FUNCTION_BLOCK CommonRack EXTENDS RunUnitGeneric
VAR_INPUT
END_VAR
VAR_OUTPUT
END_VAR
VAR
	button : POINTER TO RunSignal ;
	//TODO : define a simple output DO or DO - device?
	
	fixer : POINTER TO RunCylinder;
	approx : POINTER TO RunSignal; // approx then lock
	//---------------------------------
	//	Over Fieldbus linked with SCARA
	//---------------------------------
	rackReady AT%Q*: BOOL;
	rackEngaged AT%I*: BOOL;	

	items : ARRAY[0..3] OF defItem;
	//---------------------------------
	//	Internal
	//---------------------------------
	nCounter : INT;
END_VAR
VAR PERSISTENT
	
END_VAR


//Control the working flow of rack

SUPER^();

CASE outputState OF
	eSpecialStates.SLAVE_ENTER_PROCEDURE:
		//rack is empty
		bSerialTransition := fixer^.Execute(eCylinderCommands.COMMAND_A); //relase
		//TODO , set light flicking
	16#201:
		bSerialTransition := approx^.debouncedOn; //wait until rack closed
	16#202:
		//confirmed by hanshaking
		bSerialTransition := button^.debouncedOn;
		//TODO , set light constant on
	16#203:
		bSerialTransition := fixer^.Execute(eCylinderCommands.COMMAND_B); //lock
		IF bSerialTransition THEN
			rackReady := TRUE;
		END_IF
//		NextState := eSpecialStates.SLAVE_WORK_DONE; //release flag
	16#204:
		bSerialTransition := rackEngaged;
	16#205:
		//------------------------------------------------------------------
		//	Check if any item reached the bound. then set rackReady as false
		//------------------------------------------------------------------
		FOR nCounter := 0 TO 3 DO
			IF items[nCounter].Counter >= items[nCounter].Bound THEN
				bSerialTransition := TRUE;
				rackReady := FALSE; //released
			END_IF
		END_FOR
	16#206:
		IF NOT rackEngaged THEN
			NextState := eSpecialStates.SLAVE_ENTER_PROCEDURE; //rewind
		END_IF
END_CASE

END_FUNCTION_BLOCK

(* stored: Version 1.1.0.1, ProductVersion 3.1.4024.0
   POU CommonRack: Id {eac928e2-459d-4027-a156-266e564c65fe}, SpecialFunc None *)
